FUNCTION_BLOCK FB_TroxDrall_EL3062 IMPLEMENTS I_VolumeFlowSensor
VAR_INPUT
END_VAR
VAR_OUTPUT
END_VAR
VAR
	//Propertie Real value
	fVolumeFlow : REAL;
	//Raw value
	VolumeFlowRaw AT %I* : INT;
	//Convertion parameters
	m : REAL := 0.0444959849; //Multiplier for convertion
END_VAR

// Air Volume Flow measurement with Trox Drallauslass

PROPERTY VolumeFlow : REAL
GET
//Read volume flow
fVolumeFlow := m * INT_TO_REAL (VolumeFlowRaw); 
VolumeFlow := This^.fVolumeFlow;
END_GET
END_PROPERTY

END_FUNCTION_BLOCK

(* stored: Version 1.1.0.1
   POU FB_TroxDrall_EL3062: Id {0512a377-69d2-4887-92b7-d773adc7f8c7}, SpecialFunc None
   Property VolumeFlow: Id {27e31527-7dc0-4b40-aead-a54547972eb6}
   Get Get: Id {65686630-1534-4fe1-bb7a-fa8f0603eb9b} *)
